# EPICS StreamDevice protocol: rotating_sample_changerSup/rotsc_1.proto
#This is the protocol for the sample changer on HRPD

Terminator = '\r';
ReplyTimeout = 2000;

getID {
    out "id";
    in "%/(.{0,39})/";
	ExtraInput = Ignore;
}

getStat {
    out "st";
	in "%16s %(\$1\$2)3c %(\$1\$3)2d %(\$1\$4)2d";
	ExtraInput = Ignore;
}

getPosition {
    out "po";
	in "Position = %2d";
}

getVR {
    out "vr%(\$1\$2)#04i";
	in "%(\$1\$3){+|-} VR %*i = %i hx %*x";
	ExtraInput = Ignore;
}

sendCommand {
	out "\$1";
	in "ok";
	@mismatch {in "rf-%(\$2)i";}
}

moveWithLower {
	out "ma%#02i";
	in "ok";
	@mismatch {in "rf-%(\$1)i";}
	@init {getPosition;}
}

moveNoLower {
	out "mn%#02i";
	in "ok";
	@mismatch {in "rf-%(\$1)i";}
	@init {getPosition;}
}
